{attribute 'GeneratedUsingTerminal: EL6851-0000-0017'}
{attribute addProperty BoxType "EL6851-0000-0017"}
{attribute addProperty Id "ChannelAT %Q*ARRAY[0..63] OF USINT64"}
{attribute addProperty CRC "325009364"}
{attribute addProperty Size "64"}
TYPE DMX_Channel_DC7E3036 :
STRUCT
	{attribute addProperty Name "Channel"}
	Channel AT %Q* : ARRAY[0..63] OF USINT;
END_STRUCT
END_TYPE

(* stored: Version 1.2.0.0, ProductVersion 3.1.4024.9
   DUT DMX_Channel_DC7E3036: Id {7c3d0b3a-74bc-415f-a5b8-5a6947110a2b} *)
